FUNCTION MF_S : real
VAR_INPUT
	x,a,b:REAL;(*a defines the foot of the membership function, AND b defines its shoulder.*)

END_VAR
VAR_OUTPUT
	Error:BOOL;
END_VAR

IF NOT(b=a) THEN
	IF x<=a THEN
		MF_S := 0;
	ELSIF a<=x AND x<=(a+b)/2 THEN
		MF_S := LREAL_TO_REAL( 2*EXPT(((x-a)/(b-a)),2));
	ELSIF (a+b)/2<=x AND x<=b THEN
		MF_S := 1 - 2*LREAL_TO_REAL(EXPT(((x-b)/(b-a)),2));
	ELSIF b<=x THEN
		MF_S := 1;
	END_IF
ELSE
	Error:=TRUE;
END_IF

END_FUNCTION

(* stored: Version 1.1.0.1, ProductVersion 3.1.4024.6
   POU MF_S: Id {c5aa32e3-a1aa-4bdf-b384-9db63bd77bfb}, SpecialFunc None *)
